# EPICS autosave request: iocBoot/generic_motors_ioc/dbSave/XY_P15_.req
%
% BURT Request File
%
% $(P)XY:P15:  X-Y positioner #15
%

file assy.req ASSY=$(P)XY:P15
file mtr1.req MTR1=$(P)XY:mx15
file mtr1.req MTR1=$(P)XY:my15
file drv1.req DRV1=$(P)XY:X15
file drv1.req DRV1=$(P)XY:Y15
